# B&R Automation Studio project Sandbox
Automation Studio 4.8.3.111 SP; technology packages: mapp 5.8.0

## Configuration PC

CPU PC_any, AutomationRuntime B4.82, Build 4.1.2, Vc V4.72.1

### Task classes (Cpu.sw)
```
Cyclic#1:
  VisCtrl <- VisCtrl.prg
  Alarms <- Alarms.prg
  Count <- Count.prg
VcDataObjects: Visu <- Visu.dob
Binaries: vcctext, arialbd, vccpiech, vcmgr, vccpopup, vcxml, vccdt, vccshape, vcchspot, vcnet, vcdsloc, vcbclass, vcfntttf, Visu01, arsvcreg, vctcal, Visu03, vcshared, vcrt, vcpkat, vccbmp, TCData, vcfile, vccbtn, vccslider, vccddbox, vcalarm, vccnum, vcpdsw, FWRules, vcdsint, arial, vccovl, udbdef, vccscale, vccline, vcpdvnc, vcpfar00, vccalarm, vccstr, vcchtml, vcctrend, vcgclass, vcclbox, vccurl, Visu02, Role, arconfig, User, asfw, ashwd, ashwac, sysconf, CfgAlarm, iomap
Libraries: MpAlarmX, MpBase, astime, runtime, AsBrStr, AsARCfg, sys_lib, MpWebXs, AsArSdm
```

### Hardware
```
PC : PC_any v1.1.0.0 (OrderNumber=PC)
  Connector IF3:
    Vnc1
    VncVcObjectName1 = Visu
    VncKeyMappingFile1 = VC\PS2-Keyboard.dis
  ConfigurationID = Sandbox_PC
```

### CfgAlarm.mpalarmxcore - PC/mappServices/CfgAlarm.mpalarmxcore
```
Element gAlarmXCore (Type=mpalarmxcore)
  mapp.AlarmX.Core:
    Mapping:
      [0]:
        Alarm = CountTooHigh
        [0] = Reaction
          Name = ResetCount
  mapp.AlarmX.Core.Configuration:
    [0]:
      Name = TestAlarm
      Message = "Test Alarm!"
      Code = 10001
      Severity = 10
      Behavior = PersistentAlarm
        Acknowledge = 3
    [1]:
      Name = CountTooHigh
      Code = 10002
      Severity = 9
      Behavior = LevelMonitoring
        Acknowledge = 0
        ReactionUntilAcknowledged = FALSE
        Monitoring:
          MonitoredPV = ::Count:Count
          HighLimitEnable = Static
            Limit = 255
            LimitText = Count Too High
```

## Configuration TS_UnitTest_Sample

CPU , AutomationRuntime F4.44, Build 4.1.2

### Task classes (Cpu.sw)
```
Cyclic#4 (cycle 10000 us, tolerance 10000000 us):
  SPL_CalcTe <- TS_UnitTest.Samples.Tests_Program.Tests_MyCalcLib_C.SPL_CalcTest.prg
  SPL_CalcT1 <- TS_UnitTest.Samples.Tests_Program.Tests_MyCalcLib_C.SPL_CalcTest_Variants.prg
  SPL_Assert <- TS_UnitTest.Samples.Framework_Extension_With_Custom_Asserts.SPL_AssertsEx.prg
  SPL_Asser1 <- TS_UnitTest.Samples.Framework_Features.SPL_Asserts.prg
  SPL_Behavi <- TS_UnitTest.Samples.Framework_Features.SPL_Behavior.prg
  utTemplate <- TS_UnitTest.Templates.HelperTool_Supported.utTemplate_automated.prg
  utTemplat1 <- TS_UnitTest.Templates.NoToolSupport.utTemplate_manual.prg
Binaries: iomap, asfw, arconfig, ashwd, sysconf
Libraries: Runtime, sys_lib, AsIecCon, astime, AsARCfg, AsBrStr, UnitTest, LibAssert1, UtWs, UtMgr, SPLMyCalc
```

### Hardware
```
PC_any : PC_any v1.1.0.0 (OrderNumber=PC)
  Cyclic1Duration = 100000
  Cyclic1Tolerance = 10000000
  Cyclic2Duration = 200000
  Cyclic2Tolerance = 10000000
  Cyclic3Duration = 500000
  Cyclic3Tolerance = 10000000
  Cyclic4Duration = 10000
  Cyclic4Tolerance = 10000000
  Cyclic5Duration = 2000000
  Cyclic5Tolerance = 10000000
  Cyclic6Duration = 3000000
  Cyclic6Tolerance = 12000000
  Cyclic7Duration = 4000000
  Cyclic7Tolerance = 12000000
  Cyclic8Duration = 5000000
  Cyclic8Tolerance = 30000000
```

## Logical view

Binary libraries used (declarations not repeated): UtMgr 2.01.0, UtWs 2.01.0, operator, runtime, astime, AsIecCon, MpAlarmX 5.08.0, MpBase 5.08.0, AsBrStr, AsARCfg, sys_lib, MpWebXs 5.08.0, AsArSdm

### Global.typ - Global data types
```iecst
TYPE
	AlarmType : 	STRUCT
		Inhibit : BOOL;
		TestAlarm : BOOL;
		ResetCount : BOOL;
	END_STRUCT;
END_TYPE
```

### Global.var - Global variables
```iecst
VAR
	gAlarm : AlarmType;
END_VAR
```

### Library Logical/TS_UnitTest/Libraries/UnitTest (ANSIC, version 2.01.0) - Static library for UnitTest programs written in ANSI C /C++

#### UnitTest.h
```c
/*****************************************************************************
 * COPYRIGHT (C) BERNECKER + RAINER
 *****************************************************************************
 * Library:  UnitTest
 * File:     UnitTest.h
 * Author:   B+R
 *****************************************************************************
 * Description: Static library for UnitTest programs written in ANSI C /C++
 *
 * Add the path "\Logical\TS_UnitTest\Libraries\UnitTest\" to the
 * "Additional include directories" in the tab "Build" (PLC Properties)
 ******************************************************************************/

#ifndef	__UNITTEST_H__
#define	__UNITTEST_H__
#ifdef __cplusplus
extern "C"
{
#endif
#include <bur/plctypes.h>

#ifndef NULL
#define	NULL	0
#endif
#include "include/Test.h"

#include "include/TestCase.h"
#include "include/TestListener.h"
#include "include/TestResult.h"
#include "include/TestCaller.h"

#include "include/AssertImpl.h"
#include "include/HelperMacro.h"
#include "include/utRunner.h"

/* function is a test case */
#define _TEST 			static testStatusEnum

/* function is a setup */
#define _SETUP_TEST 	static testStatusEnum 	setupTest

/* function is a teardown */
#define _TEARDOWN_TEST 	static testStatusEnum 	teardownTest

/* function is a setup for whole test set */
#define _SETUP_SET		static testStatusEnum	setupSet

/* function is a teardown for whole test set */
#define _TEARDOWN_SET 	static testStatusEnum	teardownSet

/* function is a cyclic handler for test set */
#define _CYCLIC_SET		static void 			cyclicSetCaller

/* Skipped test case */
#define SKIP_TEST  		_TEST
/* Skip all test cases of set */
#define SKIP_TEST_SET

/* Dummies for smart edit autocompletion.
See AssertImpl.h for real macros used by the compiler  */
#ifdef _SMART_EDIT_DUMMY_

/* String comparison.
Returns true if the strings are equal. */
BOOL TEST_ASSERT_EQUAL_STRING(char *expected,char  *actual);
/* Wstring comparison.
Returns true if the WSTRINGS are equal. */
BOOL TEST_ASSERT_EQUAL_WSTRING(unsigned short *expected,unsigned short *actual);
 /* Compares two memory blocks.
Returns true if [size] bytes are equal. */
BOOL TEST_ASSERT_EQUAL_MEM(void *expected, void *actual,UDINT size);
/* Compares integer values. Usable for all integer types.
Avoid comparison of unsigned with signed types.
Returns true if they are equal.
Note: If different, values are reported as DINT values in the test report */
BOOL TEST_ASSERT_EQUAL_INT(expected, actual);

/* Compares REAL values with delta = (expected * TEST_FLOAT_PRECISION).
Returns true if (difference <= delta) */
BOOL TEST_ASSERT_EQUAL_REAL(REAL expected,REAL actual);
/* Compares REAL values with explicit delta.
Returns true if (difference <= delta) */
BOOL TEST_ASSERT_REAL_WITHIN(REAL delta, REAL expected, REAL actual);
/* Compares LREAL values with delta = (expected * TEST_DOUBLE_PRECISION).
Returns true if (difference <= delta) */
BOOL TEST_ASSERT_EQUAL_LREAL(LREAL expected,LREAL  actual);
/* Compares LREAL values with explicit delta.
Returns true if (difference <= delta) */
BOOL TEST_ASSERT_LREAL_WITHIN(LREAL delta, LREAL expected, LREAL actual);

/* Compares float values with delta = (expected * TEST_FLOAT_PRECISION).
Returns true if (difference <= delta) */
BOOL TEST_ASSERT_EQUAL_FLOAT(float expected, float actual);
/* Compares float values with explicit delta.
Returns true if (difference <= delta) */
BOOL TEST_ASSERT_FLOAT_WITHIN(float delta, float expected, float actual);
/* Compares double values with delta = (expected * TEST_DOUBLE_PRECISION).
Returns true if (difference <= delta) */
BOOL TEST_ASSERT_EQUAL_DOUBLE(double expected, double actual);
/* Compares double values with explicit delta.
Returns true if (difference <= delta) */
BOOL TEST_ASSERT_DOUBLE_WITHIN(double delta, double expected, double actual);

/* Returns true if pointer is null */
BOOL TEST_ASSERT_NULL(void *pointer);
/* Returns true if pointer is not null */
BOOL TEST_ASSERT_NOT_NULL(void *pointer);
/* Returns true, if condition evals to  true */
BOOL TEST_ASSERT_MESSAGE(condition, char *message);
/* Returns true, if condition evals to  true */
BOOL TEST_ASSERT(condition);

/* Returns always false */
BOOL TEST_FAIL(char *message);

/* Add a note to the test report */
void TEST_INFO(char *message);
/* Add a note with location information to the test report */
void TEST_INFO_POS(char *message);

#ifdef __cplusplus
/* Test if expression throws given exception.
Catches all other exceptions as failure.
Note: Available for C++ only */
void TEST_ASSERT_THROW(expression, type);

/* Fails if expression throws any exceptions.
Note: Available for C++ only*/
void TEST_ASSERT_NO_THROW(expression);
#endif

/* Adds a test function with description to the Testfixture.
See UNITTEST_FIXTURES() */
void new_TestFixture(char *name, _TEST function);

/* Adds a test function with description to the Testfixture.
This test will be skipped
See UNITTEST_FIXTURES() */
void skipTestFixture(char *name, _TEST function);

/* Defines the order of test cases.
Should look like this
UNITTEST_FIXTURES(fixtures)
{
	new_TestFixture("test_1",test_1),
	new_TestFixture("test_2",test_2),
	new_TestFixture("test_3",test_3)
}
*/
void UNITTEST_FIXTURES(fixtures)

/* Standard UnitTest caller without any setup / teardown methods*/
void UNITTEST_CALLER_TEST(caller, char *name, fixtures);

/* Standard UnitTest caller with macro setup / teardown for tests*/
void UNITTEST_CALLER_BASIC(caller, char *name, fixtures);

/* UnitTest caller with macro setup / teardown for tests and test set */
void UNITTEST_CALLER_SET(caller, char *name, fixtures);

/* UnitTest caller with macro setup / teardown for tests and test set and cylic*/
void UNITTEST_CALLER_COMPLETE(caller, char *name, fixtures);

/* UnitTest caller with explicit setup / teardown for suite */
void UNITTEST_CALLER_SET_EXPLICIT(caller,name,setupTest,teardownTest,fixtures, setupSuite, teardownSuite);

/* UnitTest caller with explicit setup / teardown for suite and cylic */
void UNITTEST_CALLER_COMPLETE_EXPLICIT(caller,name,setupTest,teardownTest,fixtures, setupSuite, teardownSuite, cyclicCaller);

/* Adds a test set with description to the fixture of test sets.
See UNITTEST_TESTSET_FIXTURES() */
void new_TestSet(testcaller);

/* Defines the order of test sets.
Should look like this
UNITTEST_TESTSET_FIXTURES(fixtures)
{
	new_TestSet(testSet_1),
	new_TestSet(testSet_2),
	new_TestSet(testSet_3)
}*/
void UNITTEST_TESTSET_FIXTURES(fixtures);

/* Defines the test set list handling structure*/
void UNTITTEST_TESTSET_HANDLER();

#endif /*_SMART_EDIT_DUMMY_*/

/*
 Use to declare Test set for use in list of test sets of test programm
 See usage in autogeneratedFile.c / FixtureOfTestSets.c
*/
#define UNITTEST_TESTSET_DECLARATION 	extern const TestCaller

/* Default factor for precision used to test if REAL / float values  are equal.
(0.00001f) */
#define TEST_FLOAT_PRECISION 	(0.00001f)
/* Default factor for precision used to test if LREAL / double values  are equal.
(1e - 12f) */
#define TEST_DOUBLE_PRECISION 	(1e-12f)

#if (__GNUC__ != 4) || (__GNUC_MINOR__ != 1) || (__GNUC_PATCHLEVEL__ != 2)
#warning UnitTest is compiled with GCC version 4.1.2. To use UnitTest switch GCC version to 4.1.2 or use different solution package
#endif

#define UNIT_TEST_LIBRARY_VERSION  			"2.01.0"

#ifdef __cplusplus
};
#endif

#include "include/asserts.hpp"

#endif/*__UNITTEST_H__*/
```

### Package Logical/TS_UnitTest/Samples/Tests_Program - Unit test sample

### Library Logical/TS_UnitTest/Samples/Tests_Program/SPLMyCalc (IEC) - Simple Calculator
Depends on: Runtime


- Program Logical/TS_UnitTest/Samples/Tests_Program/Tests_MyCalcLib_C/SPL_CalcTest (ANSIC) - Tests SPLMyCalc with library "UnitTest" (no source held here)

- Program Logical/TS_UnitTest/Samples/Tests_Program/Tests_MyCalcLib_C/SPL_CalcTest_Variants (ANSIC) - Examples how to avoid duplicated test code (advanced) (no source held here)

- Library Logical/TS_UnitTest/Samples/Framework_Extension_With_Custom_Asserts/LibAssert1 (ANSIC) - Sample library: Creation of custom asserts (no source held here)

- Program Logical/TS_UnitTest/Samples/Framework_Extension_With_Custom_Asserts/SPL_AssertsEx (ANSIC) - This sample uses custom asserts defined in LibAssert1 (no source held here)

- Program Logical/TS_UnitTest/Samples/Framework_Features/SPL_Asserts (ANSIC) - Available basic asserts (no source held here)

- Program Logical/TS_UnitTest/Samples/Framework_Features/SPL_Behavior (ANSIC) - This sample is about the control flow of test programs (no source held here)

- Program Logical/TS_UnitTest/Templates/HelperTool_Supported/utTemplate_automated (ANSIC) - Empty template for use with helper tool (no source held here)

- Program Logical/TS_UnitTest/Templates/NoToolSupport/utTemplate_manual (ANSIC) - Empty Template without support of helper tool (no source held here)

### Program Logical/UnitTests/utTestAlarm (ANSIC) - Empty template for use with helper tool

#### variables.var - Name the suite and add PVs for the program
```iecst
(********************************************************************
 * COPYRIGHT --
 ********************************************************************
 * Program: utTemplate_automated
 * File: variables.var
 * Author: -
 * Created: -
 ********************************************************************
 * Local variables of program utTemplate_automated
 ********************************************************************)
(*Describe the test*)
VAR
	Testsuite : UtMgrTestSuite := (Name:='Test Alarm',Description:='(Optional field)Template for use with helper tool. Reference or add this program in the package "TS_UnitTest_UpdateTestPrograms"',Type:=utMgrTEST_TYPE_C,MetaInformation:='(Optional field):To be filled');
END_VAR
(*Variables used in the tests*)
```

#### MappAlarmXTestAlarm.c
```c
/********************************************************************
 * COPYRIGHT --
 ********************************************************************
 * Program: -
 * Author:
 * Created:
 ********************************************************************
 * Tests for ...
 ********************************************************************/

#include <bur/plctypes.h>

#ifdef _DEFAULT_INCLUDES
#include <AsDefault.h>
#endif

#include "UnitTest.h"

_TEST WeCanTrigger(void)
{

	/* TODO:  add assertions here */

	/* test is done */
	TEST_DONE;
}
```


### Program Logical/Alarms (IEC)

#### Variables.var
```iecst
VAR
	MpAlarmXListUI_0 : MpAlarmXListUI;
	MpAlarmXCore_0 : MpAlarmXCore;
	MpAlarmXListUIConnect : MpAlarmXListUIConnectType;
END_VAR
```

#### Cyclic.st
```iecst
(*********************************************************************************
 * Copyright:
 * Author:    TylerWoodley
 * Created:   November 4, 2020/10:37 AM
 *********************************************************************************)

PROGRAM _CYCLIC
	//call the alarm FB
	MpAlarmXCore_0
	(
		Enable := TRUE,
		MpLink := ADR(gAlarmXCore)
	);
	//call the UI Link
	MpAlarmXListUI_0
	(
		MpLink := ADR(gAlarmXCore),
		Enable := TRUE,
		UIConnect := ADR(MpAlarmXListUIConnect)
	);

	//if bad thing, sound the alarm!
	IF gAlarm.TestAlarm THEN
		MpAlarmXSet(gAlarmXCore, 'TestAlarm');
	END_IF;

	//if operator is aware of bad thing, assume bad thing is handled, reset alarm.
	IF MpAlarmXCheckState(gAlarmXCore, 'TestAlarm', mpALARMX_STATE_ACKNOWLEDGED) THEN
		gAlarm.TestAlarm := FALSE;
		MpAlarmXReset(gAlarmXCore, 'TestAlarm');
	END_IF
	gAlarm.ResetCount := MpAlarmXCheckReaction(gAlarmXCore, 'ResetCount');

END_PROGRAM

PROGRAM _EXIT

		//Disable FBs
	MpAlarmXCore_0(Enable := FALSE);
	MpAlarmXListUI_0(Enable := FALSE);

END_PROGRAM
```

- Visualisation Logical/Visu (not shown)

### Program Logical/Count (IEC)

#### Cyclic.st - Cyclic code
```iecst
PROGRAM _CYCLIC
	IF gAlarm.ResetCount THEN
		Count := 0;
	ELSE
		Count := Count + 1;
	END_IF;

END_PROGRAM
```

#### Variables.var - Local variables
```iecst
VAR
	Count : USINT;
END_VAR
```

Listed in the project but not available here: Logical/TS_UnitTest/Libraries/UnitTest/include/AssertImpl.h, Logical/TS_UnitTest/Libraries/UnitTest/include/Asserts.hpp, Logical/TS_UnitTest/Libraries/UnitTest/include/HelperMacro.h, Logical/TS_UnitTest/Libraries/UnitTest/include/utRunner.h, Logical/TS_UnitTest/Libraries/UnitTest/include/Test.h, Logical/TS_UnitTest/Libraries/UnitTest/include/TestListener.h, Logical/TS_UnitTest/Libraries/UnitTest/include/TestResult.h, Logical/TS_UnitTest/Libraries/UnitTest/include/TestCaller.h, Logical/TS_UnitTest/Libraries/UnitTest/include/TestCase.h, Logical/TS_UnitTest/Samples/Tests_Program/SPLMyCalc/SPLMyCalc.typ, Logical/TS_UnitTest/Samples/Tests_Program/SPLMyCalc/SPLMyCalc.var, Logical/TS_UnitTest/Samples/Tests_Program/SPLMyCalc/SPLMyCalc.fun, Logical/TS_UnitTest/Samples/Tests_Program/SPLMyCalc/SPLMyCalc.st, Logical/TS_UnitTest/Samples/Tests_Program/Tests_MyCalcLib_C/SPL_CalcTest/variables.var, Logical/TS_UnitTest/Samples/Tests_Program/Tests_MyCalcLib_C/SPL_CalcTest/testSuite.c, Logical/TS_UnitTest/Samples/Tests_Program/Tests_MyCalcLib_C/SPL_CalcTest/autoGeneratedFile.c, Logical/TS_UnitTest/Samples/Tests_Program/Tests_MyCalcLib_C/SPL_CalcTest/testSet_MyCalcLib_Addition.c, Logical/TS_UnitTest/Samples/Tests_Program/Tests_MyCalcLib_C/SPL_CalcTest/testSet_MyCalcLib_Subtraction.c, Logical/TS_UnitTest/Samples/Tests_Program/Tests_MyCalcLib_C/SPL_CalcTest/testSet_MyCalcLib_Mult_Div.c, Logical/TS_UnitTest/Samples/Tests_Program/Tests_MyCalcLib_C/SPL_CalcTest_Variants/variables.var, Logical/TS_UnitTest/Samples/Tests_Program/Tests_MyCalcLib_C/SPL_CalcTest_Variants/testSuite.c, Logical/TS_UnitTest/Samples/Tests_Program/Tests_MyCalcLib_C/SPL_CalcTest_Variants/autoGeneratedFile.c, Logical/TS_UnitTest/Samples/Tests_Program/Tests_MyCalcLib_C/SPL_CalcTest_Variants/testSet_MyCalcLib_Subtraction.c, Logical/TS_UnitTest/Samples/Tests_Program/Tests_MyCalcLib_C/SPL_CalcTest_Variants/testSet_MyCalcLib_Subtraction_variantA.c, Logical/TS_UnitTest/Samples/Tests_Program/Tests_MyCalcLib_C/SPL_CalcTest_Variants/testSet_MyCalcLib_Subtraction_variantB.c, Logical/TS_UnitTest/Samples/Tests_Program/Tests_MyCalcLib_C/SPL_CalcTest_Variants/testSet_MyCalcLib_Subtraction_variantC.c, Logical/TS_UnitTest/Samples/Tests_Program/Tests_MyCalcLib_C/SPL_CalcTest_Variants/testSet_MyCalcLib_Subtraction_variantD.c, Logical/TS_UnitTest/Samples/Framework_Extension_With_Custom_Asserts/LibAssert1/LibAssert1.h, Logical/TS_UnitTest/Samples/Framework_Extension_With_Custom_Asserts/LibAssert1/LibAssert1_ThresholdAssert.h, Logical/TS_UnitTest/Samples/Framework_Extension_With_Custom_Asserts/LibAssert1/LibAssert1_ThresholdAssert.c, Logical/TS_UnitTest/Samples/Framework_Extension_With_Custom_Asserts/LibAssert1/LibAssert1_REAL_ArrayAsserts.h, Logical/TS_UnitTest/Samples/Framework_Extension_With_Custom_Asserts/LibAssert1/LibAssert1_REAL_ArrayAsserts.c, Logical/TS_UnitTest/Samples/Framework_Extension_With_Custom_Asserts/SPL_AssertsEx/testSuite.var, Logical/TS_UnitTest/Samples/Framework_Extension_With_Custom_Asserts/SPL_AssertsEx/testSuite.c, Logical/TS_UnitTest/Samples/Framework_Extension_With_Custom_Asserts/SPL_AssertsEx/autoGeneratedFile.c, Logical/TS_UnitTest/Samples/Framework_Extension_With_Custom_Asserts/SPL_AssertsEx/varAssertExt.var, Logical/TS_UnitTest/Samples/Framework_Extension_With_Custom_Asserts/SPL_AssertsEx/testSet_AssertsExt.c, Logical/TS_UnitTest/Samples/Framework_Features/SPL_Asserts/testSuite.var, Logical/TS_UnitTest/Samples/Framework_Features/SPL_Asserts/testSuite.c, Logical/TS_UnitTest/Samples/Framework_Features/SPL_Asserts/autoGeneratedFile.c, Logical/TS_UnitTest/Samples/Framework_Features/SPL_Asserts/varAsserts.var, Logical/TS_UnitTest/Samples/Framework_Features/SPL_Asserts/testSet_Asserts.c, Logical/TS_UnitTest/Samples/Framework_Features/SPL_Behavior/testSuite.var, Logical/TS_UnitTest/Samples/Framework_Features/SPL_Behavior/testSuite.c, Logical/TS_UnitTest/Samples/Framework_Features/SPL_Behavior/autoGeneratedFile.c, Logical/TS_UnitTest/Samples/Framework_Features/SPL_Behavior/iPrototypes.h, Logical/TS_UnitTest/Samples/Framework_Features/SPL_Behavior/iHelperFunction.h, Logical/TS_UnitTest/Samples/Framework_Features/SPL_Behavior/iHelperFunction.c, Logical/TS_UnitTest/Samples/Framework_Features/SPL_Behavior/controlFlowVariables.var, Logical/TS_UnitTest/Samples/Framework_Features/SPL_Behavior/ControlFlow/test_SetTestCases.c, Logical/TS_UnitTest/Samples/Framework_Features/SPL_Behavior/ControlFlow/test_SetTestCases_SetSetup_SetTeardown.c, Logical/TS_UnitTest/Samples/Framework_Features/SPL_Behavior/ControlFlow/test_SetTestCases_TestSetup_TestTeardown.c, Logical/TS_UnitTest/Samples/Framework_Features/SPL_Behavior/ControlFlow/test_SetComplete.c, Logical/TS_UnitTest/Samples/Framework_Features/SPL_Behavior/TestBusy_AsyncronousVariables.var, Logical/TS_UnitTest/Samples/Framework_Features/SPL_Behavior/TestBusy_Asyncronous/TestBusy_Asyncronous.c, Logical/TS_UnitTest/Samples/Framework_Features/SPL_Behavior/TestBusy_Asyncronous/TestBusy_Asyncronous_with_CyclicSet.c, Logical/TS_UnitTest/Templates/HelperTool_Supported/utTemplate_automated/variables.var, Logical/TS_UnitTest/Templates/HelperTool_Supported/utTemplate_automated/testSuite.c, Logical/TS_UnitTest/Templates/HelperTool_Supported/utTemplate_automated/autoGeneratedFile.c, Logical/TS_UnitTest/Templates/HelperTool_Supported/TestSet_Templates, Logical/TS_UnitTest/Templates/NoToolSupport/utTemplate_manual/variables.var, Logical/TS_UnitTest/Templates/NoToolSupport/utTemplate_manual/testSuite.c, Logical/TS_UnitTest/Templates/NoToolSupport/utTemplate_manual/FixtureOfTestSets.c, Logical/TS_UnitTest/Templates/NoToolSupport/TestSet_Templates/Set_Testcases.c, Logical/TS_UnitTest/Templates/NoToolSupport/TestSet_Templates/Set_SetupTeardown.c, Logical/TS_UnitTest/Templates/NoToolSupport/TestSet_Templates/Set_Complete.c, Logical/UnitTests/utTestAlarm/testSuite.c, Logical/UnitTests/utTestAlarm/autoGeneratedFile.c, Logical/VisCtrl, Logical/Count/Types.typ
